FUNCTION Convert_INT_TO_USINT : BOOL
VAR_INPUT
	in : INT;
	out : REFERENCE TO USINT;
END_VAR
VAR
	converted : USINT;
END_VAR

converted := INT_TO_USINT(in);

IF (USINT_TO_INT(converted) <> in) THEN
	RETURN;
END_IF

out := converted;
Convert_INT_TO_USINT := TRUE;

END_FUNCTION

(* stored: Version 1.1.0.1, ProductVersion 3.1.4024.12
   POU Convert_INT_TO_USINT: Id {4be41e83-b583-4dad-9099-6f958328a8b1}, SpecialFunc None *)
